% RSLogix 500 project TASK2_BAK008.RSS, saved by version 8.10.00.18 %
PROJECT "UNTITLED"    % processor: MicroLogix 1200 %

PROGRAM FILES
  LAD 2   11 rungs

DATA FILES
  O0 OUTPUT  4 elements
  I1 INPUT  4 elements
  S2 STATUS  66 elements
  B3 BINARY  1 elements
  T4 TIMER  2 elements
  C5 COUNTER  1 elements
  R6 CONTROL  1 elements
  N7 INTEGER  1 elements

LADDER 2
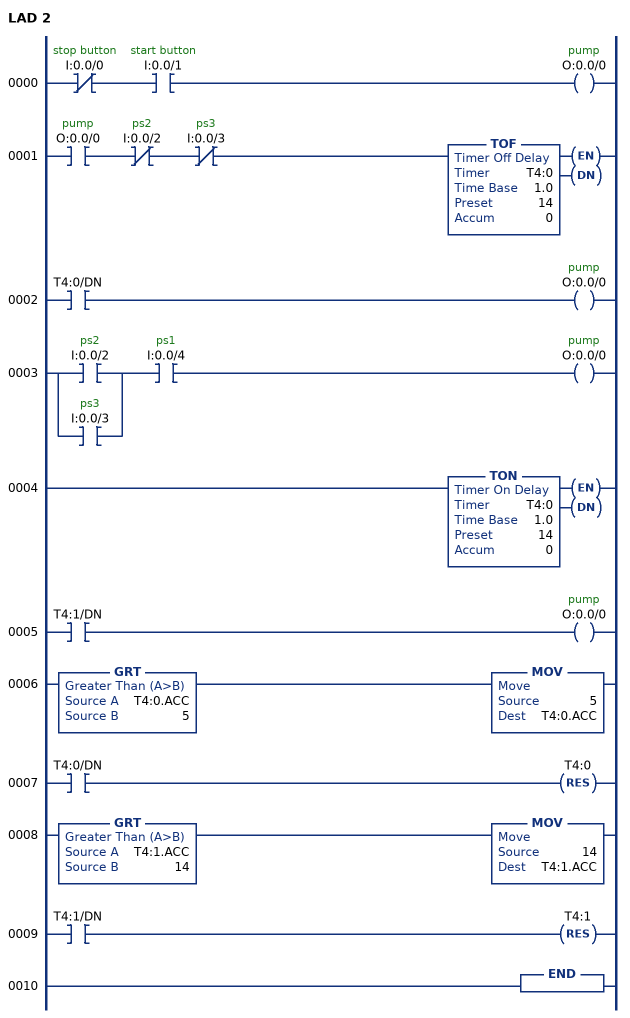
% Rung: 0 %
SOR XIO I:0.0/0 XIC I:0.0/1 OTE O:0.0/0 EOR
%   I:0.0/0  "stop button" %
%   I:0.0/1  "start button" %
%   O:0.0/0  "pump" %
% Rung: 1 %
SOR XIC O:0.0/0 XIO I:0.0/2 XIO I:0.0/3 TOF T4:0 1.0 14 0 EOR
%   O:0.0/0  "pump" %
%   I:0.0/2  "ps2" %
%   I:0.0/3  "ps3" %
% Rung: 2 %
SOR XIC T4:0/DN OTE O:0.0/0 EOR
%   O:0.0/0  "pump" %
% Rung: 3 %
SOR BST XIC I:0.0/2 NXB XIC I:0.0/3 BND XIC I:0.0/4 OTE O:0.0/0 EOR
%   I:0.0/2  "ps2" %
%   I:0.0/3  "ps3" %
%   I:0.0/4  "ps1" %
%   O:0.0/0  "pump" %
% Rung: 4 %
SOR TON T4:0 1.0 14 0 EOR
% Rung: 5 %
SOR XIC T4:1/DN OTE O:0.0/0 EOR
%   O:0.0/0  "pump" %
% Rung: 6 %
SOR GRT T4:0.ACC 5 MOV 5 T4:0.ACC EOR
% Rung: 7 %
SOR XIC T4:0/DN RES T4:0 EOR
% Rung: 8 %
SOR GRT T4:1.ACC 14 MOV 14 T4:1.ACC EOR
% Rung: 9 %
SOR XIC T4:1/DN RES T4:1 EOR
% Rung: 10 %
SOR END EOR

DATA TABLE (non-zero values as saved)
DATA T4
% .PRE .ACC %
% T4:0 % 14 0
